PROGRAM prgGrid
VAR
	FB_PV1:FB_TCPModbusRequest_Grid;
	FB_PV2:FB_TCPModbusRequest_Grid;

	lreal_GridVoltage_L1L2_V_PV1		: LREAL;				//{#lynus.ag#()}
	lreal_GridVoltage_L2L3_V_PV1		: LREAL;				//{#lynus.ag#()}
	lreal_GridVoltage_L3L1_V_PV1		: LREAL;				//{#lynus.ag#()}
	lreal_GridVoltage_L1_V_PV1			: LREAL;				//{#lynus.ag#()}
	lreal_GridVoltage_L2_V_PV1			: LREAL;				//{#lynus.ag#()}
	lreal_GridVoltage_L3_V_PV1			: LREAL;				//{#lynus.ag#()}
	lreal_GridCurrent_L1_A_PV1			: LREAL;				//{#lynus.ag#()}
	lreal_GridCurrent_L2_A_PV1			: LREAL;				//{#lynus.ag#()}
	lreal_GridCurrent_L3_A_PV1			: LREAL;				//{#lynus.ag#()}
	lreal_GridPower_kW_PV1				: LREAL;				//{#lynus.ag#()}
	lreal_GridReactivePower_kVAr_PV1	: LREAL;				//{#lynus.ag#()}
	lreal_GridPowerFactor_PV1			: LREAL;				//{#lynus.ag#()}
	lreal_GridFrequency_Hz_PV1			: LREAL;				//{#lynus.ag#()}
	lreal_GridEnergyDelivered_kWh_PV1	: LREAL;				//{#lynus.ag#()}
	lreal_GridEnergySupllied_kWh_PV1	: LREAL;				//{#lynus.ag#()}
	
	lreal_GridVoltage_L1L2_V_PV2		: LREAL;				//{#lynus.ag#()}
	lreal_GridVoltage_L2L3_V_PV2		: LREAL;				//{#lynus.ag#()}
	lreal_GridVoltage_L3L1_V_PV2		: LREAL;				//{#lynus.ag#()}
	lreal_GridVoltage_L1_V_PV2			: LREAL;				//{#lynus.ag#()}
	lreal_GridVoltage_L2_V_PV2			: LREAL;				//{#lynus.ag#()}
	lreal_GridVoltage_L3_V_PV2			: LREAL;				//{#lynus.ag#()}
	lreal_GridCurrent_L1_A_PV2			: LREAL;				//{#lynus.ag#()}
	lreal_GridCurrent_L2_A_PV2			: LREAL;				//{#lynus.ag#()}
	lreal_GridCurrent_L3_A_PV2			: LREAL;				//{#lynus.ag#()}
	lreal_GridPower_kW_PV2				: LREAL;				//{#lynus.ag#()}
	lreal_GridReactivePower_kVAr_PV2	: LREAL;				//{#lynus.ag#()}
	lreal_GridPowerFactor_PV2			: LREAL;				//{#lynus.ag#()}
	lreal_GridFrequency_Hz_PV2			: LREAL;				//{#lynus.ag#()}
	lreal_GridEnergyDelivered_kWh_PV2	: LREAL;				//{#lynus.ag#()}
	lreal_GridEnergySupllied_kWh_PV2	: LREAL;				//{#lynus.ag#()}

	lreal_HousePower_kW_PV1				: LREAL;				//{#lynus.ag#()}
	lreal_HousePower_kW_PV2				: LREAL;				//{#lynus.ag#()}

END_VAR


FB_PV1	(	b_Enable:= TRUE, 
			str_IPAdress:= prgPv.FB_PV1.str_IPAdress);


FB_PV2	(	b_Enable:= TRUE, 
			str_IPAdress:= prgPv.FB_PV2.str_IPAdress);



lreal_GridVoltage_L1L2_V_PV1 	:= FB_PV1.lreal_GridVoltage_L1L2_V;
lreal_GridVoltage_L2L3_V_PV1 	:= FB_PV1.lreal_GridVoltage_L2L3_V;
lreal_GridVoltage_L3L1_V_PV1 	:= FB_PV1.lreal_GridVoltage_L3L1_V;
lreal_GridVoltage_L1_V_PV1		:= FB_PV1.lreal_GridVoltage_L1_V;
lreal_GridVoltage_L2_V_PV1		:= FB_PV1.lreal_GridVoltage_L2_V;
lreal_GridVoltage_L3_V_PV1		:= FB_PV1.lreal_GridVoltage_L3_V;
lreal_GridCurrent_L1_A_PV1		:= FB_PV1.lreal_GridCurrent_L1_A;
lreal_GridCurrent_L2_A_PV1		:= FB_PV1.lreal_GridCurrent_L2_A;
lreal_GridCurrent_L3_A_PV1		:= FB_PV1.lreal_GridCurrent_L3_A;
lreal_GridPower_kW_PV1			:= FB_PV1.lreal_GridPower_kW;
lreal_GridReactivePower_kVAr_PV1:= FB_PV1.lreal_GridReactivePower_kVAr;
lreal_GridPowerFactor_PV1		:= FB_PV1.lreal_GridPowerFactor;
lreal_GridFrequency_Hz_PV1		:= FB_PV1.lreal_GridFrequency_Hz;
lreal_GridEnergyDelivered_kWh_PV1:= FB_PV1.lreal_GridEnergyDelivered_kWh;
lreal_GridEnergySupllied_kWh_PV1 := FB_PV1.lreal_GridEnergySupllied_kWh;

lreal_HousePower_kW_PV1 := lreal_GridPower_kW_PV1 + prgPV.lrPowerPV1;

lreal_GridVoltage_L1L2_V_PV2 	:= FB_PV2.lreal_GridVoltage_L1L2_V;
lreal_GridVoltage_L2L3_V_PV2 	:= FB_PV2.lreal_GridVoltage_L2L3_V;
lreal_GridVoltage_L3L1_V_PV2 	:= FB_PV2.lreal_GridVoltage_L3L1_V;
lreal_GridVoltage_L1_V_PV2		:= FB_PV2.lreal_GridVoltage_L1_V;
lreal_GridVoltage_L2_V_PV2		:= FB_PV2.lreal_GridVoltage_L2_V;
lreal_GridVoltage_L3_V_PV2		:= FB_PV2.lreal_GridVoltage_L3_V;
lreal_GridCurrent_L1_A_PV2		:= FB_PV2.lreal_GridCurrent_L1_A;
lreal_GridCurrent_L2_A_PV2		:= FB_PV2.lreal_GridCurrent_L2_A;
lreal_GridCurrent_L3_A_PV2		:= FB_PV2.lreal_GridCurrent_L3_A;
lreal_GridPower_kW_PV2			:= FB_PV2.lreal_GridPower_kW;
lreal_GridReactivePower_kVAr_PV2:= FB_PV2.lreal_GridReactivePower_kVAr;
lreal_GridPowerFactor_PV2		:= FB_PV2.lreal_GridPowerFactor;
lreal_GridFrequency_Hz_PV2		:= FB_PV2.lreal_GridFrequency_Hz;
lreal_GridEnergyDelivered_kWh_PV2:= FB_PV2.lreal_GridEnergyDelivered_kWh;
lreal_GridEnergySupllied_kWh_PV2 := FB_PV2.lreal_GridEnergySupllied_kWh;


lreal_HousePower_kW_PV2 := lreal_GridPower_kW_PV1 + prgPV.lrPowerPV2;

END_PROGRAM

(* stored: Version 1.1.0.1, ProductVersion 3.1.4024.11
   POU prgGrid: Id {9da87431-0904-45b1-a35c-2d3365b9066c}, SpecialFunc None *)
